// TIA Portal V17 export
// export: Created 2024-08-26T21:07:18.3895788Z, ExportSetting WithDefaults, DisplayName Totally Integrated Automation Portal, DisplayVersion V17 Update 7, DisplayName TIA Portal Openness, DisplayVersion V17 Update 7, DisplayName TIA Portal Version Control Interface, DisplayVersion V17, DisplayName SINAMICS Startdrive Advanced, DisplayVersion V17 SP2, DisplayName SINAMICS Startdrive G110M, G120, G120C, G120D, G120P, G115D, DisplayVersion V17 SP2, DisplayName SINAMICS Startdrive G130, G150, S120, S150, SINAMICS MV, S210, DisplayVersion V17 SP2, DisplayName STEP 7 Professional, DisplayVersion V17 Update 7, DisplayName STEP 7 Safety, DisplayVersion V17 Update 6, DisplayName WinCC Advanced / Unified PC, DisplayVersion V17 Update 7
FUNCTION "production" : Void   // FC15, LAD
{ S7_Optimized_Access := 'TRUE' }
VERSION : 0.1
// stored: AutoNumber true, IsIECCheckEnabled false, SetENOAutomatically false, UDAEnableTagReadback false
   VAR_TEMP   // added for the SCL form of the ladder/FBD networks
      _w1 : Bool;
      _w2 : Bool;
      _w3 : Bool;
   END_VAR
BEGIN

REGION Network 1: SHIFTS PRODUCTION
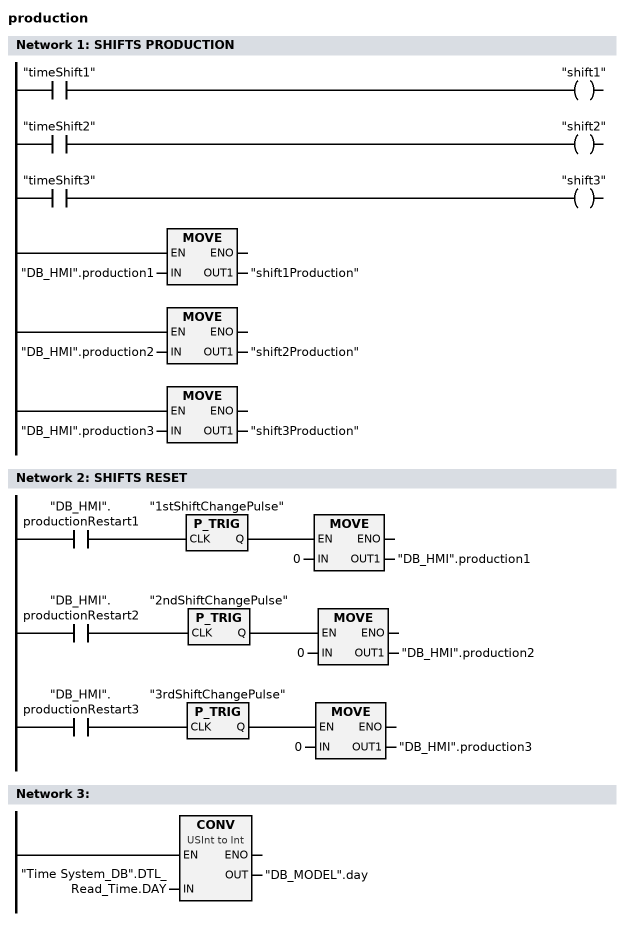
   RUNG wire#powerrail
      Contact( "timeShift1" )
      Coil( "shift1" )
   END_RUNG
   RUNG wire#powerrail
      Contact( "timeShift2" )
      Coil( "shift2" )
   END_RUNG
   RUNG wire#powerrail
      Contact( "timeShift3" )
      Coil( "shift3" )
   END_RUNG
   RUNG wire#powerrail
      Move(in := "DB_HMI".production1, out1 => "shift1Production")
   END_RUNG
   RUNG wire#powerrail
      Move(in := "DB_HMI".production2, out1 => "shift2Production")
   END_RUNG
   RUNG wire#powerrail
      Move(in := "DB_HMI".production3, out1 => "shift3Production")
   END_RUNG
   // the same network as SCL:
   "shift1" := "timeShift1";
   "shift2" := "timeShift2";
   "shift3" := "timeShift3";
   "shift1Production" := "DB_HMI".production1;
   "shift2Production" := "DB_HMI".production2;
   "shift3Production" := "DB_HMI".production3;
END_REGION

REGION Network 2: SHIFTS RESET
   RUNG wire#powerrail
      Contact( "DB_HMI".productionRestart1 )
      P_Trig( "1stShiftChangePulse" )
      Move(in := 0, out1 => "DB_HMI".production1)
   END_RUNG
   RUNG wire#powerrail
      Contact( "DB_HMI".productionRestart2 )
      P_Trig( "2ndShiftChangePulse" )
      Move(in := 0, out1 => "DB_HMI".production2)
   END_RUNG
   RUNG wire#powerrail
      Contact( "DB_HMI".productionRestart3 )
      P_Trig( "3rdShiftChangePulse" )
      Move(in := 0, out1 => "DB_HMI".production3)
   END_RUNG
   // the same network as SCL:
   #_w1 := "DB_HMI".productionRestart1 AND NOT "1stShiftChangePulse";   // rising edge
   "1stShiftChangePulse" := "DB_HMI".productionRestart1;
   IF #_w1 THEN "DB_HMI".production1 := 0; END_IF;
   #_w2 := "DB_HMI".productionRestart2 AND NOT "2ndShiftChangePulse";   // rising edge
   "2ndShiftChangePulse" := "DB_HMI".productionRestart2;
   IF #_w2 THEN "DB_HMI".production2 := 0; END_IF;
   #_w3 := "DB_HMI".productionRestart3 AND NOT "3rdShiftChangePulse";   // rising edge
   "3rdShiftChangePulse" := "DB_HMI".productionRestart3;
   IF #_w3 THEN "DB_HMI".production3 := 0; END_IF;
END_REGION

REGION Network 3
   RUNG wire#powerrail
      { S7_Templates := "[SrcType := USInt, DestType := Int]" } Convert(in := "Time System_DB".DTL_Read_Time.DAY, out => "DB_MODEL".day)
   END_RUNG
   // the same network as SCL:
   "DB_MODEL".day := USINT_TO_INT("Time System_DB".DTL_Read_Time.DAY);
END_REGION
END_FUNCTION
